Fanuc KAREL source: IO0007.KL

-- PROVISIONAL review KL for V770-1; original PC SHA256 af83c08f1b137117bede3bbdd4c1093f4346fa19accaf095caf5e42f6ba4619f
-- Incomplete behavior may be omitted. Consult companion uncertainty JSON. Do not deploy.
PROGRAM IO0007
%NOLOCKGROUP
-- UNRESOLVED_LOCAL_POOL 5 cells at code offset 13; source declarations unknown
-- DIRECT_LOCAL_WORD_ACCESS alone does not prove INTEGER, REAL, or BOOLEAN
BEGIN
  -- UNRESOLVED_PC offsets 0-18; opcodes 2B,2C,7B
  -- UNRESOLVED_PC offsets 23-30; opcodes 9D,23
  -- UNRESOLVED_PC offsets 35-49; opcodes 2E,22,9D,33,35
  -- UNRESOLVED_PC offsets 54-61; opcodes 9D,23
  -- UNRESOLVED_PC offsets 66-77; opcodes 2E,23
  -- UNRESOLVED_PC offsets 82-96; opcodes 21,19,23
  -- UNRESOLVED_PC offsets 101-105; opcodes 7F
  -- UNRESOLVED_PC offsets 110-114; opcodes 27,AA
  -- UNRESOLVED_PC offsets 119-123; opcodes 7F
END IO0007
